// TIA Portal V17 export
// export: Created 2025-03-13T10:30:29.8665202Z, ExportSetting WithDefaults, DisplayName Totally Integrated Automation Portal, DisplayVersion V17 Update 8, DisplayName TIA Portal Openness, DisplayVersion V17 Update 8, DisplayName TIA Portal Version Control Interface, DisplayVersion V17, DisplayName SINAMICS Startdrive Advanced, DisplayVersion V17 SP2, DisplayName SINAMICS Startdrive G110M, G120, G120C, G120D, G120P, G115D, DisplayVersion V17 SP2, DisplayName SINAMICS Startdrive G130, G150, S120, S150, SINAMICS MV, S210, DisplayVersion V17 SP2, DisplayName STEP 7 Professional, DisplayVersion V17 Update 8, DisplayName SINUMERIK ONE STEP 7 Toolbox, DisplayVersion V17 Update 12, DisplayName SINUMERIK 840D sl STEP 7 Toolbox, DisplayVersion V17 Update 12, DisplayName STEP 7 Safety, DisplayVersion V17 Update 6, DisplayName WinCC Advanced, DisplayVersion V17 Update 8
DATA_BLOCK "DB2401_DBB_DEFINE"   // DB2401
{ S7_Optimized_Access := 'FALSE'; DB_Accessible_From_OPC_UA := 'FALSE' }
AUTHOR : ETXETAR
VERSION : 1.0
// stored: AutoNumber false, DBAccessibleFromOPCUA false, DBAccessibleFromWebserver true, IsOnlyStoredInLoadMemory false, IsWriteProtectedInAS false
   VAR RETAIN
      DBB_0 : Byte;   // MACHINE CNC CYCLE UNIT 01 STATION 0 STATION 1
      DBB_1 : Byte;
      DBB_2 : Byte;   // MACHINE CNC CYCLE UNIT 01 STATION 3
      DBB_3 : Byte;
      DBB_4 : Byte;   // MACHINE CNC CYCLE UNIT 01 STATION 4
      DBB_5 : Byte;
      DBB_6 : Byte;   // MACHINE CNC CYCLE UNIT 02 STATION 0 STATION 1
      DBB_7 : Byte;
      DBB_8 : Byte;   // MACHINE CNC CYCLE UNIT 02 STATION 2
      DBB_9 : Byte;
      DBB_10 : Byte;   // MACHINE CNC CYCLE UNIT 02 STATION 3
      DBB_11 : Byte;
      DBB_12 : Byte;   // MACHINE CNC CYCLE UNIT 02 STATION 4
      DBB_13 : Byte;
      DBB_14 : Byte;   // MACHINE CNC CYCLE UNIT 03
      DBB_15 : Byte;
      DBB_16 : Byte;
      DBB_17 : Byte;
      DBB_18 : Byte;
      DBB_19 : Byte;
      DBB_20 : Byte;   // FIXTURE NUMBER IN UNIT 01 STATION 1
      DBB_21 : Byte;
      DBB_22 : Byte;   // FIXTURE NUMBER IN UNIT 02 STATION 1
      DBB_23 : Byte;
      DBB_24 : Byte;
      DBB_25 : Byte;
      DBW_26 : Int;
      DBW_28 : Int;
      DBB_30 : Byte;   // PART TYPE
      DBB_31 : Byte;
      DBB_32 : Byte;
      DBB_33 : Byte;
      DBB_34 : Byte;
      DBB_35 : Byte;
      DBB_36 : Byte;
      DBB_37 : Byte;
      DBW_38 : Int;
      DBB_40 : Byte;   // FIXTURE 1 MACHINING MEMORY TO FULL DEPTH UNIT 01R
      DBB_41 : Byte;   // FIXTURE 1 MACHINING MEMORY TO FULL DEPTH UNIT 01L
      DBB_42 : Byte;
      DBB_43 : Byte;
      DBB_44 : Byte;   // FIXTURE 1 BACK CHAMFERS TRACER
      DBB_45 : Byte;   // FIXTURE 1 TAPPING TRACER
      DBB_46 : Byte;
      DBB_47 : Byte;
      DBB_48 : Byte;   // FIXTURE 2 MACHINING MEMORY TO FULL DEPTH UNIT 01R
      DBB_49 : Byte;   // FIXTURE 2 MACHINING MEMORY TO FULL DEPTH UNIT 01L
      DBB_50 : Byte;
      DBB_51 : Byte;
      DBB_52 : Byte;   // FIXTURE 2 BACK CHAMFERS TRACER
      DBB_53 : Byte;   // FIXTURE 2 TAPPING TRACER
      DBB_54 : Byte;
      DBB_55 : Byte;
      DBB_56 : Byte;   // FIXTURE 1 CLAMP STATUS
      DBB_57 : Byte;   // FIXTURE 2 CLAMP STATUS
      DBB_58 : Byte;   // PART SEATED CLAMP RECOVERY UNIT 01R
      DBB_59 : Byte;   // PART SEATED CLAMP RECOVERY UNIT 01L
      DBB_60 : Byte;   // AXIS W SAFETY MOVE
      DBB_61 : Byte;   // AXIS B POSITIONS
      DBB_62 : Byte;   // AXIS B IN POSITION TO LOAD
      DBB_63 : Byte;
      DBB_64 : Byte;   // MEASURE PROBE ALARM CODE
      DBB_65 : Byte;   // MEASUREMENT FRECUENCY
      DBB_66 : Byte;   // RESET GUD CYCLE VARIABLES
      DBB_67 : Byte;   // CYCLE SELECTION CEMB ENABLE
      DBB_68 : Byte;
      DBB_69 : Byte;
      DBB_70 : Byte;   // MQL VARIANT UNIT 01R
      DBB_71 : Byte;   // MQL VARIANT UNIT 01L
      DBB_72 : Byte;
      DBB_73 : Byte;
      DBB_74 : Byte;
      DBB_75 : Byte;   // RFID ZONE TO WRITE IN TOOL HOLDER CHIP UNIT 01R
      DBB_76 : Byte;   // RFID ZONE TO WRITE IN TOOL HOLDER CHIP UNIT 01L
      DBB_77 : Byte;   // RFID ZONE TO WRITE IN TOOL HOLDER CHIP
      DBB_78 : Byte;
      DBB_79 : Byte;
      DBB_80 : Byte;   // TAG ERROR UNIT 01R
      DBB_81 : Byte;   // TAG ERROR UNIT 01L
      DBB_82 : Byte;
      DBB_83 : Byte;
      DBB_84 : Byte;
      SPARE_86 : Array[1..14] of Byte;
      DBB_100 : Byte;   // TOOL CLAMPING DIFFERENCE SP11
      DBB_101 : Byte;   // TOOL CLAMPING DIFFERENCE SP12
      DBB_102 : Byte;   // TOOL CLAMPING DIFFERENCE SP13
      DBB_103 : Byte;   // TOOL CLAMPING DIFFERENCE SP14
      SPARE_104 : Array[1..6] of Byte;
      DBB_110 : Byte;   // TOOL CLAMPING DIFFERENCE SP21
      DBB_111 : Byte;   // TOOL CLAMPING DIFFERENCE SP22
      DBB_112 : Byte;   // TOOL CLAMPING DIFFERENCE SP23
      DBB_113 : Byte;   // TOOL CLAMPING DIFFERENCE SP24
      SPARE_114 : Array[1..6] of Byte;
      DBB_120 : Byte;   // MAGAZINE MEMORY ALARM UNIT 01R
      DBB_121 : Byte;   // MAGAZINE MEMORY ALARM TYPE UNIT 01R
      DBB_122 : Byte;   // MAGAZINE TOOL FAULTED UNIT 01R
      DBB_123 : Byte;   // MAGAZINE TOOL IN ERROR DATA UNIT 01R
      DBB_124 : Byte;
      DBB_125 : Byte;   // MAGAZINE MEMORY ALARM UNIT 01L
      DBB_126 : Byte;   // MAGAZINE MEMORY ALARM TYPE UNIT 01L
      DBB_127 : Byte;   // MAGAZINE TOOL FAULTED UNIT 01L
      DBB_128 : Byte;   // MAGAZINE TOOL IN ERROR DATA UNIT 01L
      DBB_129 : Byte;
      DBB_130 : Byte;
      DBB_131 : Byte;
      DBB_132 : Byte;
      DBB_133 : Byte;
      DBB_134 : Byte;
      SPARE_136 : Array[1..14] of Byte;
      DBB_150 : Byte;   // BK MIKRO MAGAZINE POSITION SP11
      DBB_151 : Byte;   // BK MIKRO MAGAZINE POSITION SP12
      DBB_152 : Byte;   // BK MIKRO MAGAZINE POSITION SP13
      DBB_153 : Byte;   // BK MIKRO MAGAZINE POSITION SP14
      DBB_154 : Byte;   // BK MIKRO MAGAZINE POSITION SP21
      DBB_155 : Byte;   // BK MIKRO MAGAZINE POSITION SP22
      DBB_156 : Byte;   // BK MIKRO MAGAZINE POSITION SP23
      DBB_157 : Byte;   // BK MIKRO MAGAZINE POSITION SP24
      DBB_158 : Byte;
      DBB_159 : Byte;
      DBR_160 : Real;   // UNIT 01 POWDER FEEDER 1 CARRIER GAS NOMINAL LINE 1
      DBR_164 : Real;   // UNIT 01 POWDER FEEDER 1 CARRIER GAS NOMINAL LINE 2
      DBR_168 : Real;   // UNIT 01 POWDER FEEDER 1 DISK SPEED NOMINAL LINE 1
      DBR_172 : Real;   // UNIT 01 POWDER FEEDER 1 DISK SPEED NOMINAL LINE 2
      DBR_176 : Real;   // UNIT 01 POWDER FEEDER 1 STIRRER SPEED NOMINAL LINE 1
      DBR_180 : Real;   // UNIT 01 POWDER FEEDER 1 STIRRER SPEED NOMINAL LINE 2
      DBR_184 : Real;   // UNIT 01 POWDER FEEDER 1 HOPPER TEMPERATURE NOMINAL LINE 1
      DBR_188 : Real;   // UNIT 01 POWDER FEEDER 1 HOPPER TEMPERATURE NOMINAL LINE 2
      SPARE_192 : Array[192..199] of Byte;
      DBR_200 : Real;   // UNIT 02 POWDER FEEDER 1 CARRIER GAS NOMINAL LINE 1
      DBR_204 : Real;   // UNIT 02 POWDER FEEDER 1 CARRIER GAS NOMINAL LINE 2
      DBR_208 : Real;   // UNIT 02 POWDER FEEDER 1 DISK SPEED NOMINAL LINE 1
      DBR_212 : Real;   // UNIT 02 POWDER FEEDER 1 DISK SPEED NOMINAL LINE 2
      DBR_216 : Real;   // UNIT 02 POWDER FEEDER 1 STIRRER SPEED NOMINAL LINE 1
      DBR_220 : Real;   // UNIT 02 POWDER FEEDER 1 STIRRER SPEED NOMINAL LINE 2
      DBR_224 : Real;   // UNIT 02 POWDER FEEDER 1 HOPPER TEMPERATURE NOMINAL LINE 1
      DBR_228 : Real;   // UNIT 02 POWDER FEEDER 1 HOPPER TEMPERATURE NOMINAL LINE 2
      SPARE_232 : Array[232..239] of Byte;
      DBR_240 : Real;   // UNIT 02 POWDER FEEDER 2 CARRIER GAS NOMINAL LINE 1
      DBR_244 : Real;   // UNIT 02 POWDER FEEDER 2 CARRIER GAS NOMINAL LINE 2
      DBR_248 : Real;   // UNIT 02 POWDER FEEDER 2 DISK SPEED NOMINAL LINE 1
      DBR_252 : Real;   // UNIT 02 POWDER FEEDER 2 DISK SPEED NOMINAL LINE 2
      DBR_256 : Real;   // UNIT 02 POWDER FEEDER 2 STIRRER SPEED NOMINAL LINE 1
      DBR_260 : Real;   // UNIT 02 POWDER FEEDER 2 STIRRER SPEED NOMINAL LINE 2
      DBR_264 : Real;   // UNIT 02 POWDER FEEDER 2 HOPPER TEMPERATURE NOMINAL LINE 1
      DBR_268 : Real;   // UNIT 02 POWDER FEEDER 2 HOPPER TEMPERATURE NOMINAL LINE 2
      SPARE_272 : Array[272..503] of Byte;
      DBW_504 : Word;   // UNIT 01 LASER POWER
      DBW_506 : Word;   // UNIT 01 LASER PROCESSING (0=CORE / 1=RING / 3=BRIGHTLINE WELD)
      DBW_508 : Word;   // UNIT 01 LASER POWER PORTION CORE (%)
      DBB_510 : Byte;
      DBB_511 : Byte;
      DBB_512 : Byte;
      DBB_513 : Byte;
      DBW_514 : Word;   // UNIT 02 LASER POWER
      DBW_516 : Word;   // UNIT 02 LASER PROCESSING (0=CORE / 1=RING / 3=BRIGHTLINE WELD)
      DBW_518 : Word;   // UNIT 02 LASER POWER PORTION CORE (%)
      SPARE_520 : Array[520..999] of Byte;
      PART_STATUS : Struct   // PART STATUS
         DBB_1000 : Byte;   // UNIT 01 FIXTURE 1 PART A QUALITY STATUS
         DBB_1001 : Byte;   // UNIT 01 FIXTURE 1 PART A PROCESS STATUS
         DBB_1002 : Byte;   // UNIT 01 FIXTURE 1 PART C
         DBB_1003 : Byte;   // UNIT 01 FIXTURE 1 PART D
         DBB_1004 : Byte;
         DBB_1005 : Byte;
         DBB_1006 : Byte;   // UNIT 01 FIXTURE 2 PART A QUALITY STATUS
         DBB_1007 : Byte;   // UNIT 01 FIXTURE 2 PART A PROCESS STATUS
         DBB_1008 : Byte;   // UNIT 01 FIXTURE 2 PART C
         DBB_1009 : Byte;   // UNIT 01 FIXTURE 2 PART D
         DBB_1010 : Byte;
         DBB_1011 : Byte;
         DBB_1012 : Byte;   // UNIT 01 FIXTURE 3 PART A QUALITY STATUS
         DBB_1013 : Byte;   // UNIT 01 FIXTURE 3 PART A PROCESS STATUS
         DBB_1014 : Byte;   // UNIT 01 FIXTURE 3 PART C
         DBB_1015 : Byte;   // UNIT 01 FIXTURE 3 PART D
         DBB_1016 : Byte;
         DBB_1017 : Byte;
         DBB_1018 : Byte;   // UNIT 01 FIXTURE 4 PART A QUALITY STATUS
         DBB_1019 : Byte;   // UNIT 01 FIXTURE 4 PART A PROCESS STATUS
         DBB_1020 : Byte;   // UNIT 01 FIXTURE 4 PART C
         DBB_1021 : Byte;   // UNIT 01 FIXTURE 4 PART D
         DBB_1022 : Byte;
         DBB_1023 : Byte;
         DBB_1024 : Byte;   // UNIT 02 FIXTURE 1 PART A QUALITY STATUS
         DBB_1025 : Byte;   // UNIT 02 FIXTURE 1 PART A PROCESS STATUS
         DBB_1026 : Byte;   // UNIT 02 FIXTURE 1 PART C
         DBB_1027 : Byte;   // UNIT 02 FIXTURE 1 PART D
         DBB_1028 : Byte;
         DBB_1029 : Byte;
         DBB_1030 : Byte;   // UNIT 02 FIXTURE 2 PART A QUALITY STATUS
         DBB_1031 : Byte;   // UNIT 02 FIXTURE 2 PART A PROCESS STATUS
         DBB_1032 : Byte;   // UNIT 02 FIXTURE 2 PART C
         DBB_1033 : Byte;   // UNIT 02 FIXTURE 2 PART D
         DBB_1034 : Byte;
         DBB_1035 : Byte;
         DBB_1036 : Byte;   // UNIT 02 FIXTURE 3 PART A QUALITY STATUS
         DBB_1037 : Byte;   // UNIT 02 FIXTURE 3 PART A PROCESS STATUS
         DBB_1038 : Byte;   // UNIT 02 FIXTURE 3 PART C
         DBB_1039 : Byte;   // UNIT 02 FIXTURE 3 PART D
         DBB_1040 : Byte;
         DBB_1041 : Byte;
         DBB_1042 : Byte;   // UNIT 02 FIXTURE 4 PART A QUALITY STATUS
         DBB_1043 : Byte;   // UNIT 02 FIXTURE 4 PART A PROCESS STATUS
         DBB_1044 : Byte;   // UNIT 02 FIXTURE 4 PART C
         DBB_1045 : Byte;   // UNIT 02 FIXTURE 4 PART D
         DBB_1046 : Byte;
         DBB_1047 : Byte;
         DBB_1048 : Byte;   // UNIT 01 STATION 1 PART A QUALITY STATUS
         DBB_1049 : Byte;   // UNIT 01 STATION 1 PART A PROCESS STATUS
         DBB_1050 : Byte;   // UNIT 01 STATION 1 PART C
         DBB_1051 : Byte;   // UNIT 01 STATION 1 PART D
         DBB_1052 : Byte;
         DBB_1053 : Byte;
         DBB_1054 : Byte;   // UNIT 01 STATION 2 PART A QUALITY STATUS
         DBB_1055 : Byte;   // UNIT 01 STATION 2 PART A PROCESS STATUS
         DBB_1056 : Byte;   // UNIT 01 STATION 2 PART C
         DBB_1057 : Byte;   // UNIT 01 STATION 2 PART D
         DBB_1058 : Byte;
         DBB_1059 : Byte;
         DBB_1060 : Byte;   // UNIT 01 STATION 3 PART A QUALITY STATUS
         DBB_1061 : Byte;   // UNIT 01 STATION 3 PART A PROCESS STATUS
         DBB_1062 : Byte;   // UNIT 01 STATION 3 PART C
         DBB_1063 : Byte;   // UNIT 01 STATION 3 PART D
         DBB_1064 : Byte;
         DBB_1065 : Byte;
         DBB_1066 : Byte;   // UNIT 01 STATION 4 PART A QUALITY STATUS
         DBB_1067 : Byte;   // UNIT 01 STATION 4 PART A PROCESS STATUS
         DBB_1068 : Byte;   // UNIT 01 STATION 4 PART C
         DBB_1069 : Byte;   // UNIT 01 STATION 4 PART D
         DBB_1070 : Byte;
         DBB_1071 : Byte;
         DBB_1072 : Byte;   // UNIT 02 STATION 1 PART A QUALITY STATUS
         DBB_1073 : Byte;   // UNIT 02 STATION 1 PART A PROCESS STATUS
         DBB_1074 : Byte;   // UNIT 02 STATION 1 PART C
         DBB_1075 : Byte;   // UNIT 02 STATION 1 PART D
         DBB_1076 : Byte;
         DBB_1077 : Byte;
         DBB_1078 : Byte;   // UNIT 02 STATION 2 PART A QUALITY STATUS
         DBB_1079 : Byte;   // UNIT 02 STATION 2 PART A PROCESS STATUS
         DBB_1080 : Byte;   // UNIT 02 STATION 2 PART C
         DBB_1081 : Byte;   // UNIT 02 STATION 2 PART D
         DBB_1082 : Byte;
         DBB_1083 : Byte;
         DBB_1084 : Byte;   // UNIT 02 STATION 3 PART A QUALITY STATUS
         DBB_1085 : Byte;   // UNIT 02 STATION 3 PART A PROCESS STATUS
         DBB_1086 : Byte;   // UNIT 02 STATION 3 PART C
         DBB_1087 : Byte;   // UNIT 02 STATION 3 PART D
         DBB_1088 : Byte;
         DBB_1089 : Byte;
         DBB_1090 : Byte;   // UNIT 02 STATION 4 PART A QUALITY STATUS
         DBB_1091 : Byte;   // UNIT 02 STATION 4 PART A PROCESS STATUS
         DBB_1092 : Byte;   // UNIT 02 STATION 4 PART C
         DBB_1093 : Byte;   // UNIT 02 STATION 4 PART D
         DBB_1094 : Byte;
         DBB_1095 : Byte;
         DBB_1096 : Byte;   // UNIT 03 FIXTURE 1 PART A QUALITY STATUS
         DBB_1097 : Byte;   // UNIT 03 FIXTURE 1 PART A PROCESS STATUS
         DBB_1098 : Byte;   // UNIT 03 FIXTURE 1 PART C
         DBB_1099 : Byte;   // UNIT 01 FIXTURE 1 PART D
         DBB_1100 : Byte;
      END_STRUCT;
      SPARE_1102 : Array[48..145] of Byte;
      DBB_1200 : Byte;   // CLEAN TOOL HOLDERS UNIT 01R
      DBB_1201 : Byte;   // CLEAN TOOL HOLDERS SEQUENCE DONE UNIT 01R
      DBB_1202 : Byte;
      DBB_1203 : Byte;
      DBB_1204 : Byte;   // CLEAN TOOL HOLDERS UNIT 01L
      DBB_1205 : Byte;   // CLEAN TOOL HOLDERS SEQUENCE DONE UNIT 01L
      DBB_1206 : Byte;
      DBB_1207 : Byte;
      DBB_1208 : Byte;
      DBB_1209 : Byte;
      SPARE_1210 : Array[1..39] of Byte;
      DBW_1250 : Int;   // WAIT CHANNEL 1
      SPARE_1252 : Array[1..20] of Byte;
      DBR_1272 : Real;   // UNIT 01 AXIS X13 ACTUAL SPEED
      DBR_1276 : Real;   // UNIT 01 AXIS Z13 ACTUAL SPEED
      DBR_1280 : Real;   // UNIT 01 AXIS E10 ACTUAL SPEED
      DBR_1284 : Real;   // UNIT 01 SPINDLE C11 ACTUAL SPEED
      DBR_1288 : Real;   // UNIT 01 SPINDLE C12 ACTUAL SPEED
      DBR_1292 : Real;   // UNIT 01 SPINDLE C13 ACTUAL SPEED
      DBR_1296 : Real;   // UNIT 01 SPINDLE C14 ACTUAL SPEED
      DBR_1300 : Real;   // UNIT 01 PROCESS SETPOINT SPEED
      DBR_1304 : Real;
      SPARE_1308 : Array[1..44] of Byte;
      DBR_1352 : Real;   // UNIT 02 AXIS X23 ACTUAL SPEED
      DBR_1356 : Real;   // UNIT 02 AXIS Z23 ACTUAL SPEED
      DBR_1360 : Real;   // UNIT 02 AXIS E20 ACTUAL SPEED
      DBR_1364 : Real;   // UNIT 02 SPINDLE C21 ACTUAL SPEED
      DBR_1368 : Real;   // UNIT 02 SPINDLE C22 ACTUAL SPEED
      DBR_1372 : Real;   // UNIT 02 SPINDLE C23 ACTUAL SPEED
      DBR_1376 : Real;   // UNIT 02 SPINDLE C24 ACTUAL SPEED
      DBR_1380 : Real;   // UNIT 02 PROCESS SETPOINT SPEED
      SPARE_1384 : Array[1..66] of Byte;
      DBW_1450 : Int;   // NC TEST PROGRAM AXIS SELECTION
      DBW_1452 : Int;   // SERVICE POSITION PROGRAM SELECTION
      DBW_1454 : Int;   // SPEED FOR SP11. VIBRATION ANALYSIS
      DBW_1456 : Int;   // SPEED FOR SP12. VIBRATION ANALYSIS
      DBW_1458 : Int;   // TIME FOR ANALYSIS. VIBRATION ANALYSIS UNIT 01R
      DBW_1460 : Int;   // TIME FOR START. VIBRATION ANALYSIS UNIT 01R
      DBW_1462 : Int;   // SPEED FOR SP21. VIBRATION ANALYSIS
      DBW_1464 : Int;   // SPEED FOR SP22. VIBRATION ANALYSIS
      DBW_1466 : Int;   // TIME FOR ANALYSIS. VIBRATION ANALYSIS UNIT 01L
      DBW_1468 : Int;   // TIME FOR START. VIBRATION ANALYSIS UNIT 01L
      SPARE_1470 : Array[1..30] of Byte;
      TOOL_NAME_01R : Array[1..32] of Char;   // TOOL NAME. TOOL MAGAZINE 01R
      DBW_1532 : Int;   // DUPLO NUMBER. TOOL MAGAZINE 01R
      DBW_1534 : Int;   // LOCATION TYPE. TOOL MAGAZINE 01R
      DBW_1536 : Int;   // SIEMENS TOOL STATUS. TOOL MAGAZINE 01R
      DBW_1538 : Int;   // TYPE OF TOOL MONITORING. TOOL MAGAZINE 01R
      DBW_1540 : Int;   // CHECK TOOL BROKEN. TOOL MAGAZINE 01R
      DBW_1542 : Int;   // NUMBER OF CUTTING EDGES. TOOL MAGAZINE 01R
      DBD_1544 : DInt;   // OEM 1. TOOL MAGAZINE 01R
      DBR_1548 : Real;   // OEM 2. TOOL MAGAZINE 01R
      DBR_1552 : Real;   // OEM 3. TOOL MAGAZINE 01R
      DBR_1556 : Real;   // OEM 4. TOOL MAGAZINE 01R
      DBR_1560 : Real;   // OEM 5. TOOL MAGAZINE 01R
      DBR_1564 : Real;   // OEM 6. TOOL MAGAZINE 01R
      DBR_1568 : Real;   // OEM 7. TOOL MAGAZINE 01R
      DBR_1572 : Real;   // OEM 8. TOOL MAGAZINE 01R
      DBR_1576 : Real;   // OEM 9. TOOL MAGAZINE 01R
      DBR_1580 : Real;   // OEM 10. TOOL MAGAZINE 01R
      DBW_1584 : Int;   // TOOL TYPE EDGE 1. TOOL MAGAZINE 01R
      DBW_1586 : Int;   // CUTTING POSITION EDGE 1. TOOL MAGAZINE 01R
      DBR_1588 : Real;   // TOOL LENGTH 1 EDGE 1. TOOL MAGAZINE 01R
      DBR_1592 : Real;   // TOOL LENGTH 2 EDGE 1. TOOL MAGAZINE 01R
      DBR_1596 : Real;   // TOOL LENGTH 3 EDGE 1. TOOL MAGAZINE 01R
      DBR_1600 : Real;   // TOOL RADIUS EDGE 1. TOOL MAGAZINE 01R
      DBR_1604 : Real;   // TOOL PITCH EDGE 1. TOOL MAGAZINE 01R
      DBR_1608 : Real;   // WEAR LENGTH EDGE 1. TOOL MAGAZINE 01R
      DBR_1612 : Real;
      DBR_1616 : Real;
      DBR_1620 : Real;   // WEAR RADIUS EDGE 1. TOOL MAGAZINE 01R
      DBR_1624 : Real;
      DBR_1628 : Real;
      DBR_1632 : Real;
      DBR_1636 : Real;
      DBR_1640 : Real;
      DBR_1644 : Real;   // WARNING TOOL LIFE EDGE 1. TOOL MAGAZINE 01R
      DBR_1648 : Real;   // ACTUAL TOOL LIFE EDGE 1. TOOL MAGAZINE 01R
      DBR_1652 : Real;   // SET POINT QUANTITY EDGE 1. TOOL MAGAZINE 01R
      DBR_1656 : Real;
      DBR_1660 : Real;
      DBW_1664 : Int;   // TOOL TYPE EDGE 2. TOOL MAGAZINE 01R
      DBW_1666 : Int;   // CUTTING POSITION EDGE 2. TOOL MAGAZINE 01R
      DBR_1668 : Real;   // TOOL LENGTH 1 EDGE 2. TOOL MAGAZINE 01R
      DBR_1672 : Real;   // TOOL LENGTH 2 EDGE 2. TOOL MAGAZINE 01R
      DBR_1676 : Real;   // TOOL LENGTH 3 EDGE 2. TOOL MAGAZINE 01R
      DBR_1680 : Real;   // TOOL RADIUS EDGE 2. TOOL MAGAZINE 01R
      DBR_1684 : Real;   // TOOL PITCH EDGE 2. TOOL MAGAZINE 01R
      DBR_1688 : Real;   // WEAR LENGTH EDGE 2. TOOL MAGAZINE 01R
      DBR_1692 : Real;
      DBR_1696 : Real;
      DBR_1700 : Real;   // UNIT 01 NOZZLE SURFACE DISTANCE
      DBR_1704 : Real;   // UNIT 02 NOZZLE SURFACE DISTANCE
      DBR_1708 : Real;
      DBR_1712 : Real;
      DBR_1716 : Real;
      DBR_1720 : Real;
      DBR_1724 : Real;   // WARNING TOOL LIFE EDGE 2. TOOL MAGAZINE 01R
      DBR_1728 : Real;   // ACTUAL TOOL LIFE EDGE 2. TOOL MAGAZINE 01R
      DBR_1732 : Real;   // SET POINT QUANTITY EDGE 2. TOOL MAGAZINE 01R
      DBR_1736 : Real;
      DBR_1740 : Real;
      DBW_1744 : Int;   // TOOL TYPE EDGE 3. TOOL MAGAZINE 01R
      DBW_1746 : Int;   // CUTTING POSITION EDGE 3. TOOL MAGAZINE 01R
      DBR_1748 : Real;   // TOOL LENGTH 1 EDGE 3. TOOL MAGAZINE 01R
      DBR_1752 : Real;   // TOOL LENGTH 2 EDGE 3. TOOL MAGAZINE 01R
      DBR_1756 : Real;   // TOOL LENGTH 3 EDGE 3. TOOL MAGAZINE 01R
      DBR_1760 : Real;   // TOOL RADIUS EDGE 3. TOOL MAGAZINE 01R
      DBR_1764 : Real;   // TOOL PITCH EDGE 3. TOOL MAGAZINE 01R
      DBR_1768 : Real;   // WEAR LENGTH EDGE 3. TOOL MAGAZINE 01R
      DBR_1772 : Real;
      DBR_1776 : Real;
      DBR_1780 : Real;   // WEAR RADIUS EDGE 3. TOOL MAGAZINE 01R
      DBR_1784 : Real;
      DBR_1788 : Real;
      DBR_1792 : Real;
      DBR_1796 : Real;
      DBR_1800 : Real;
      DBR_1804 : Real;   // WARNING TOOL LIFE EDGE 3. TOOL MAGAZINE 01R
      DBR_1808 : Real;   // ACTUAL TOOL LIFE EDGE 3. TOOL MAGAZINE 01R
      DBR_1812 : Real;   // SET POINT QUANTITY EDGE 3. TOOL MAGAZINE 01R
      DBR_1816 : Real;
      DBR_1820 : Real;
      DBW_1824 : Int;   // TOOL TYPE EDGE 4. TOOL MAGAZINE 01R
      DBW_1826 : Int;   // CUTTING POSITION EDGE 4. TOOL MAGAZINE 01R
      DBR_1828 : Real;   // TOOL LENGTH 1 EDGE 4. TOOL MAGAZINE 01R
      DBR_1832 : Real;   // TOOL LENGTH 2 EDGE 4. TOOL MAGAZINE 01R
      DBR_1836 : Real;   // TOOL LENGTH 3 EDGE 4. TOOL MAGAZINE 01R
      DBR_1840 : Real;   // TOOL RADIUS EDGE 4. TOOL MAGAZINE 01R
      DBR_1844 : Real;   // TOOL PITCH EDGE 4. TOOL MAGAZINE 01R
      DBR_1848 : Real;   // WEAR LENGTH EDGE 4. TOOL MAGAZINE 01R
      DBR_1852 : Real;
      DBR_1856 : Real;
      DBR_1860 : Real;   // WEAR RADIUS EDGE 4. TOOL MAGAZINE 01R
      DBR_1864 : Real;
      DBR_1868 : Real;
      DBR_1872 : Real;
      DBR_1876 : Real;
      DBR_1880 : Real;
      DBR_1884 : Real;   // WARNING TOOL LIFE EDGE 4. TOOL MAGAZINE 01R
      DBR_1888 : Real;   // ACTUAL TOOL LIFE EDGE 4. TOOL MAGAZINE 01R
      DBR_1892 : Real;   // SET POINT QUANTITY EDGE 4. TOOL MAGAZINE 01R
      DBR_1896 : Real;
      DBR_1900 : Real;
      DBW_1904 : Int;   // TOOL TYPE EDGE 5. TOOL MAGAZINE 01R
      DBW_1906 : Int;   // CUTTING POSITION EDGE 5. TOOL MAGAZINE 01R
      DBR_1908 : Real;   // TOOL LENGTH 1 EDGE 5. TOOL MAGAZINE 01R
      DBR_1912 : Real;   // TOOL LENGTH 2 EDGE 5. TOOL MAGAZINE 01R
      DBR_1916 : Real;   // TOOL LENGTH 3 EDGE 5. TOOL MAGAZINE 01R
      DBR_1920 : Real;   // TOOL RADIUS EDGE 5. TOOL MAGAZINE 01R
      DBR_1924 : Real;   // TOOL PITCH EDGE 5. TOOL MAGAZINE 01R
      DBR_1928 : Real;   // WEAR LENGTH EDGE 5. TOOL MAGAZINE 01R
      DBR_1932 : Real;
      DBR_1936 : Real;
      DBR_1940 : Real;   // WEAR RADIUS EDGE 5. TOOL MAGAZINE 01R
      DBR_1944 : Real;
      DBR_1948 : Real;
      DBR_1952 : Real;
      DBR_1956 : Real;
      DBR_1960 : Real;
      DBR_1964 : Real;   // WARNING TOOL LIFE EDGE 5. TOOL MAGAZINE 01R
      DBR_1968 : Real;   // ACTUAL TOOL LIFE EDGE 5. TOOL MAGAZINE 01R
      DBR_1972 : Real;   // SET POINT QUANTITY EDGE 5. TOOL MAGAZINE 01R
      DBR_1976 : Real;
      DBR_1980 : Real;
      DBB_1984 : Byte;   // GM SPINDLE NUMBER 01R
      SPARE_1986 : Array[1..14] of Byte;
      TOOL_NAME_01L : Array[1..32] of Char;   // TOOL NAME. TOOL MAGAZINE 01L
      DBW_2032 : Int;   // DUPLO NUMBER. TOOL MAGAZINE 01L
      DBW_2034 : Int;   // LOCATION TYPE. TOOL MAGAZINE 01L
      DBW_2036 : Int;   // SIEMENS TOOL STATUS. TOOL MAGAZINE 01L
      DBW_2038 : Int;   // TYPE OF TOOL MONITORING. TOOL MAGAZINE 01L
      DBW_2040 : Int;   // CHECK TOOL BROKEN. TOOL MAGAZINE 01L
      DBW_2042 : Int;   // NUMBER OF CUTTING EDGES. TOOL MAGAZINE 01L
      DBD_2044 : DInt;   // OEM 1. TOOL MAGAZINE 01L
      DBR_2048 : Real;   // OEM 2. TOOL MAGAZINE 01L
      DBR_2052 : Real;   // OEM 3. TOOL MAGAZINE 01L
      DBR_2056 : Real;   // OEM 4. TOOL MAGAZINE 01L
      DBR_2060 : Real;   // OEM 5. TOOL MAGAZINE 01L
      DBR_2064 : Real;   // OEM 6. TOOL MAGAZINE 01L
      DBR_2068 : Real;   // OEM 7. TOOL MAGAZINE 01L
      DBR_2072 : Real;   // OEM 8. TOOL MAGAZINE 01L
      DBR_2076 : Real;   // OEM 9. TOOL MAGAZINE 01L
      DBR_2080 : Real;   // OEM 10. TOOL MAGAZINE 01L
      DBW_2084 : Int;   // TOOL TYPE EDGE 1. TOOL MAGAZINE 01L
      DBW_2086 : Int;   // CUTTING POSITION EDGE 1. TOOL MAGAZINE 01L
      DBR_2088 : Real;   // TOOL LENGTH 1 EDGE 1. TOOL MAGAZINE 01L
      DBR_2092 : Real;   // TOOL LENGTH 2 EDGE 1. TOOL MAGAZINE 01L
      DBR_2096 : Real;   // TOOL LENGTH 3 EDGE 1. TOOL MAGAZINE 01L
      DBR_2100 : Real;   // TOOL RADIUS EDGE 1. TOOL MAGAZINE 01L
      DBR_2104 : Real;   // TOOL PITCH EDGE 1. TOOL MAGAZINE 01L
      DBR_2108 : Real;   // WEAR LENGTH EDGE 1. TOOL MAGAZINE 01L
      DBR_2112 : Real;
      DBR_2116 : Real;
      DBR_2120 : Real;   // WEAR RADIUS EDGE 1. TOOL MAGAZINE 01L
      DBR_2124 : Real;
      DBR_2128 : Real;
      DBR_2132 : Real;
      DBR_2136 : Real;
      DBR_2140 : Real;
      DBR_2144 : Real;   // WARNING TOOL LIFE EDGE 1. TOOL MAGAZINE 01L
      DBR_2148 : Real;   // ACTUAL TOOL LIFE EDGE 1. TOOL MAGAZINE 01L
      DBR_2152 : Real;   // SET POINT QUANTITY EDGE 1. TOOL MAGAZINE 01L
      DBR_2156 : Real;
      DBR_2160 : Real;
      DBW_2164 : Int;   // TOOL TYPE EDGE 2. TOOL MAGAZINE 01L
      DBW_2166 : Int;   // CUTTING POSITION EDGE 2. TOOL MAGAZINE 01L
      DBR_2168 : Real;   // TOOL LENGTH 1 EDGE 2. TOOL MAGAZINE 01L
      DBR_2172 : Real;   // TOOL LENGTH 2 EDGE 2. TOOL MAGAZINE 01L
      DBR_2176 : Real;   // TOOL LENGTH 3 EDGE 2. TOOL MAGAZINE 01L
      DBR_2180 : Real;   // TOOL RADIUS EDGE 2. TOOL MAGAZINE 01L
      DBR_2184 : Real;   // TOOL PITCH EDGE 2. TOOL MAGAZINE 01L
      DBR_2188 : Real;   // WEAR LENGTH EDGE 2. TOOL MAGAZINE 01L
      DBR_2192 : Real;
      DBR_2196 : Real;
      DBR_2200 : Real;   // WEAR RADIUS EDGE 2. TOOL MAGAZINE 01L
      DBR_2204 : Real;
      DBR_2208 : Real;
      DBR_2212 : Real;
      DBR_2216 : Real;
      DBR_2220 : Real;
      DBR_2224 : Real;   // WARNING TOOL LIFE EDGE 2. TOOL MAGAZINE 01L
      DBR_2228 : Real;   // ACTUAL TOOL LIFE EDGE 2. TOOL MAGAZINE 01L
      DBR_2232 : Real;   // SET POINT QUANTITY EDGE 2. TOOL MAGAZINE 01L
      DBR_2236 : Real;
      DBR_2240 : Real;
      DBW_2244 : Int;   // TOOL TYPE EDGE 3. TOOL MAGAZINE 01L
      DBW_2246 : Int;   // CUTTING POSITION EDGE 3. TOOL MAGAZINE 01L
      DBR_2248 : Real;   // TOOL LENGTH 1 EDGE 3. TOOL MAGAZINE 01L
      DBR_2252 : Real;   // TOOL LENGTH 2 EDGE 3. TOOL MAGAZINE 01L
      DBR_2256 : Real;   // TOOL LENGTH 3 EDGE 3. TOOL MAGAZINE 01L
      DBR_2260 : Real;   // TOOL RADIUS EDGE 3. TOOL MAGAZINE 01L
      DBR_2264 : Real;   // TOOL PITCH EDGE 3. TOOL MAGAZINE 01L
      DBR_2268 : Real;   // WEAR LENGTH EDGE 3. TOOL MAGAZINE 01L
      DBR_2272 : Real;
      DBR_2276 : Real;
      DBR_2280 : Real;   // WEAR RADIUS EDGE 3. TOOL MAGAZINE 01L
      DBR_2284 : Real;
      DBR_2288 : Real;
      DBR_2292 : Real;
      DBR_2296 : Real;
      DBR_2300 : Real;
      DBR_2304 : Real;   // WARNING TOOL LIFE EDGE 3. TOOL MAGAZINE 01L
      DBR_2308 : Real;   // ACTUAL TOOL LIFE EDGE 3. TOOL MAGAZINE 01L
      DBR_2312 : Real;   // SET POINT QUANTITY EDGE 3. TOOL MAGAZINE 01L
      DBR_2316 : Real;
      DBR_2320 : Real;
      DBW_2324 : Int;   // TOOL TYPE EDGE 4. TOOL MAGAZINE 01L
      DBW_2326 : Int;   // CUTTING POSITION EDGE 4. TOOL MAGAZINE 01L
      DBR_2328 : Real;   // TOOL LENGTH 1 EDGE 4. TOOL MAGAZINE 01L
      DBR_2332 : Real;   // TOOL LENGTH 2 EDGE 4. TOOL MAGAZINE 01L
      DBR_2336 : Real;   // TOOL LENGTH 3 EDGE 4. TOOL MAGAZINE 01L
      DBR_2340 : Real;   // TOOL RADIUS EDGE 4. TOOL MAGAZINE 01L
      DBR_2344 : Real;   // TOOL PITCH EDGE 4. TOOL MAGAZINE 01L
      DBR_2348 : Real;   // WEAR LENGTH EDGE 4. TOOL MAGAZINE 01L
      DBR_2352 : Real;
      DBR_2356 : Real;
      DBR_2360 : Real;   // WEAR RADIUS EDGE 4. TOOL MAGAZINE 01L
      DBR_2364 : Real;
      DBR_2368 : Real;
      DBR_2372 : Real;
      DBR_2376 : Real;
      DBR_2380 : Real;
      DBR_2384 : Real;   // WARNING TOOL LIFE EDGE 4. TOOL MAGAZINE 01L
      DBR_2388 : Real;   // ACTUAL TOOL LIFE EDGE 4. TOOL MAGAZINE 01L
      DBR_2392 : Real;   // SET POINT QUANTITY EDGE 4. TOOL MAGAZINE 01L
      DBR_2396 : Real;
      DBR_2400 : Real;
      DBW_2404 : Int;   // TOOL TYPE EDGE 5. TOOL MAGAZINE 01L
      DBW_2406 : Int;   // CUTTING POSITION EDGE 5. TOOL MAGAZINE 01L
      DBR_2408 : Real;   // TOOL LENGTH 1 EDGE 5. TOOL MAGAZINE 01L
      DBR_2412 : Real;   // TOOL LENGTH 2 EDGE 5. TOOL MAGAZINE 01L
      DBR_2416 : Real;   // TOOL LENGTH 3 EDGE 5. TOOL MAGAZINE 01L
      DBR_2420 : Real;   // TOOL RADIUS EDGE 5. TOOL MAGAZINE 01L
      DBR_2424 : Real;   // TOOL PITCH EDGE 5. TOOL MAGAZINE 01L
      DBR_2428 : Real;   // WEAR LENGTH EDGE 5. TOOL MAGAZINE 01L
      DBR_2432 : Real;
      DBR_2436 : Real;
      DBR_2440 : Real;   // WEAR RADIUS EDGE 5. TOOL MAGAZINE 01L
      DBR_2444 : Real;
      DBR_2448 : Real;
      DBR_2452 : Real;
      DBR_2456 : Real;
      DBR_2460 : Real;
      DBR_2464 : Real;   // WARNING TOOL LIFE EDGE 5. TOOL MAGAZINE 01L
      DBR_2468 : Real;   // ACTUAL TOOL LIFE EDGE 5. TOOL MAGAZINE 01L
      DBR_2472 : Real;   // SET POINT QUANTITY EDGE 5. TOOL MAGAZINE 01L
      DBR_2476 : Real;
      DBR_2480 : Real;
      DBB_2484 : Byte;   // GM SPINDLE NUMBER 01L
      SPARE_2486 : Array[1..514] of Byte;
      DBR_3000 : Real;   // CRASH BORE MEASURE POINT 1
      DBR_3004 : Real;   // CRASH BORE MEASURE POINT 2
      DBR_3008 : Real;   // CRASH BORE MEASURE POINT 3
      DBR_3012 : Real;   // CRASH BORE MEASURE POINT 4
      DBR_3016 : Real;   // CRASH BORE MEASURE POINT 5
      DBR_3020 : Real;   // CRASH BORE MEASURE POINT 6
      DBR_3024 : Real;   // CRASH BORE MEASURE POINT 7X
      DBR_3028 : Real;   // CRASH BORE MEASURE POINT 7Y
      DBR_3032 : Real;   // CRASH BORE MEASURE POINT 8X
      DBR_3036 : Real;   // CRASH BORE MEASURE POINT 8Y
      SPARE_3040 : Array[1..160] of Byte;
      DBR_3200 : Real;   // MEASURING PROBE PART A 1
      DBR_3204 : Real;   // MEASURING PROBE PART A 2
      DBR_3208 : Real;   // MEASURING PROBE PART B 1
      DBR_3212 : Real;   // MEASURING PROBE PART B 2
      DBR_3216 : Real;   // MEASURING PROBE PART C 1
      DBR_3220 : Real;   // MEASURING PROBE PART C 2
      DBR_3224 : Real;   // MEASURING PROBE PART A1 1
      DBR_3228 : Real;   // MEASURING PROBE PART A1 2
      DBR_3232 : Real;   // MEASURING PROBE PART B1 1
      DBR_3236 : Real;   // MEASURING PROBE PART B1 2
      DBR_3240 : Real;   // MEASURING PROBE PART C1 1
      DBR_3244 : Real;   // MEASURING PROBE PART C1 2
      DBR_3248 : Real;   // MEASURING PROBE PART A2 1
      DBR_3252 : Real;   // MEASURING PROBE PART A2 2
      DBR_3256 : Real;   // MEASURING PROBE PART B2 1
      DBR_3260 : Real;   // MEASURING PROBE PART B2 2
      DBR_3264 : Real;   // MEASURING PROBE PART C2 1
      DBR_3268 : Real;   // MEASURING PROBE PART C2 2
      SPARE_3272 : Array[1..128] of Byte;
      DBR_3400 : Real;   // TORQUE AXIS SP11
      DBR_3404 : Real;   // TORQUE AXIS SP12
      DBR_3408 : Real;   // TORQUE AXIS SP13
      DBR_3412 : Real;   // TORQUE AXIS SP14
      DBR_3416 : Real;   // TORQUE AXIS SP15
      DBR_3420 : Real;   // TORQUE AXIS SP16
      DBR_3424 : Real;   // TORQUE AXIS SP21
      DBR_3428 : Real;   // TORQUE AXIS SP22
      DBR_3432 : Real;   // TORQUE AXIS SP23
      DBR_3436 : Real;   // TORQUE AXIS SP24
      DBR_3440 : Real;   // TORQUE AXIS SP25
      DBR_3444 : Real;   // TORQUE AXIS SP26
      DBR_3448 : Real;   // TORQUE AXIS Z11
      DBR_3452 : Real;   // TORQUE AXIS Z12
      DBR_3456 : Real;   // TORQUE AXIS Z13
      DBR_3460 : Real;   // TORQUE AXIS Z14
      DBR_3464 : Real;   // TORQUE AXIS Z21
      DBR_3468 : Real;   // TORQUE AXIS Z22
      DBR_3472 : Real;   // TORQUE AXIS Z23
      DBR_3476 : Real;   // TORQUE AXIS Z24
      SPARE_3480 : Array[1..520] of Byte;
   END_VAR
BEGIN
END_DATA_BLOCK
